PROGRAM pCounter
VAR
	fbCTU: CTU;
	bSW1 AT %I*: BOOL;
	bSW2 AT %I*: BOOL;
	CurrentValue: WORD;
	bLED1 AT %Q*: BOOL;
END_VAR

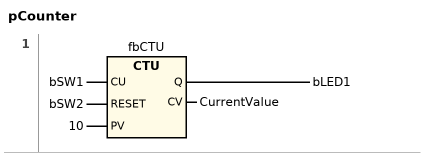
// NETWORK 1
fbCTU(CU := bSW1, RESET := bSW2, PV := 10, CV => CurrentValue); // CTU
bLED1 := fbCTU.Q;

END_PROGRAM

(* stored: Version 1.1.0.1, ProductVersion 3.1.4024.2
   POU pCounter: Id {85f9cfb1-5ad3-4c1a-8579-d3cfb95c2742}, SpecialFunc None *)
